Yaskawa INFORM job: PLACE-RECTANGLE.JBI

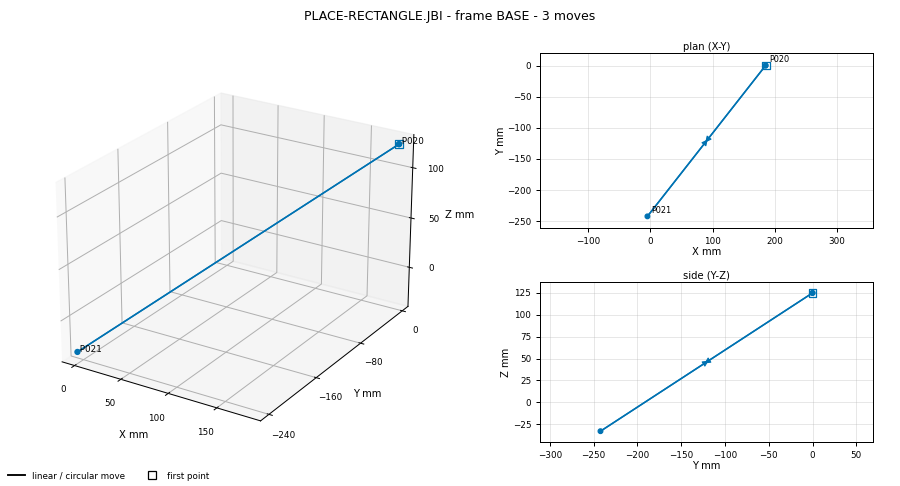
[picture p0: tool path of PLACE-RECTANGLE.JBI in frame BASE, 3 of 3 moves have a stored position in this frame; points joined in program order, loops and branches not executed]
/JOB
//NAME PLACE-RECTANGLE
//POS
///NPOS 0,0,0,3,0,0
///TOOL 0
///POSTYPE BASE
///RECTAN
///RCONF 1,0,0,0,0,0,0,0,0,0,0,0,0,0,0,0,0,0,0,0,0,0,0,0
P00020=185.000,0.000,125.000,180.0000,0.0000,0.0000
P00021=-4.816,-242.273,-32.953,-179.9759,-2.4091,-91.1631
P00022=185.001,0.012,125.015,-179.9824,-0.0082,0.0088
//INST
///DATE 2019/05/19 12:33
///ATTR SC,RW
///GROUP1 RB1
NOP
MOVL P020 V=187.0
MOVL P021 V=187.0
DOUT OT#(1) OFF
MOVL P022 V=187.0
RET
END
